TYPE ZONA_OUTPUT :
	STRUCT
		LIBERO     : BOOL := FALSE;
		TRIGGER    : BOOL := FALSE;
	END_STRUCT
END_TYPE

(* stored: Version 1.1.0.1, ProductVersion 3.1.4024.12
   DUT ZONA_OUTPUT: Id {ad704a6a-187d-469c-a08d-883bc1c302a9} *)
